(* PLC project OOP_Curso, Beckhoff Automation GmbH TwinCAT PLC Control 3.5.13.21 *)
(* stored: creationDateTime 2023-04-01T13:18:38.4462117, modificationDateTime 2023-04-01T13:18:38.451092 *)

FUNCTION_BLOCK FB_1 EXTENDS FB_Base
VAR_OUTPUT
    nBase: INT;
END_VAR

            THIS^.METH_DoIt();      // llamada al metodo METH_DoIt del FB_1.
THIS^.METH_DoAlso();

SUPER^.METH_DoIt();     // llamada al metodo METH_DoIt del FB_Base.
SUPER^.METH_DoAlso();
nBase := SUPER^.nCnt;
          

METHOD METH_DoAlso : BOOL
                  nCnt := 123;    
METH_DoAlso := FALSE;
                
END_METHOD

METHOD METH_DoIt : BOOL
                  nCnt := 1111;    
METH_DoIt := TRUE;
                
END_METHOD
END_FUNCTION_BLOCK

FUNCTION_BLOCK FB_Base
VAR_OUTPUT
    nCnt : INT;
END_VAR

            
          

METHOD METH_DoAlso : BOOL
VAR_INPUT
END_VAR
                  METH_DoAlso := TRUE;
                
END_METHOD

METHOD METH_DoIt : BOOL
                  nCnt := -1;
                
END_METHOD
END_FUNCTION_BLOCK

FUNCTION F_FunA : INT
VAR_INPUT
    fbMyFbA : FB_A;
END_VAR

            
          
END_FUNCTION

FUNCTION_BLOCK FB_A
VAR_INPUT
    nVarA: INT;
END_VAR

            nVarA := 1;
          
END_FUNCTION_BLOCK

FUNCTION_BLOCK FB_B EXTENDS FB_A
VAR_INPUT
    nVarB : INT := 0;
END_VAR

            nVarA := 11;
nVarB := 2;
          

METHOD DoIt : BOOL
VAR_INPUT
END_VAR
VAR
    nVarB : INT;
END_VAR
                  nVarB := 22; // Se establece la variable local nVarB.
THIS^.nVarB := 222; // La variable del bloque de funciones nVarB se establece aunque nVarB está oculta.
F_FunA(fbMyFbA := THIS^);  //F_FunA es llamado via THIS^.
                
END_METHOD
END_FUNCTION_BLOCK

PROGRAM _09_THIS_SUPER
VAR
	// Ejemplo para el puntero THIS^
	fbMyfbB : FB_B;
	
	// Ejemplo para el puntero SUPER^
    fbMyBase : FB_Base;
    fbMyFB_1 : FB_1;
    nTHIS    : INT;
    nBase    : INT;	
END_VAR

            // Ejemplo para el puntero THIS^
fbMyfbB(nVarA:=0, nVarB:= 0);
fbMyfbB.DoIt();

// Ejemplo para el puntero SUPER^
fbMyBase();
nBase := fbmyBase.nCnt;
fbMyFB_1();
nTHIS := fbMyFB_1.nCnt;
          
END_PROGRAM
